(* Logix 5000 project; controller Laser_Cutter vendor 1 type 14 code 149 rev 28.11; software revision 28.00; part 4 of 4 *)
(* tags used below, declared in another part *)
   aAcceptPartSol : BOOL;
   aBlowOffOnSol : BOOL;
   aBoltBowlFeedingOn : BOOL;
   aBoltDriverDownSol : BOOL;
   aBoltDriverForward : BOOL;
   aBoltDriverReverse : BOOL;
   aBoltDriverUpSol : BOOL;
   aBoltFeedingTrackOn : BOOL;
   aCameraTrigger : BOOL;
   acceptPartSol : BOOL;
   aClampingStation2Down : BOOL;
   aClampingStation2Up : BOOL;
   aClampingStation4DownSol : BOOL;
   aClampingStation5DownSol : BOOL;
   aClampingStation5UpSol : BOOL;
   aCollarBowlFeedingOn : BOOL;
   aCollarFeedingTrackOn : BOOL;
   aDoorSafetySwitchUnlockSol : BOOL;
   alarmActive : BOOL;
   aRejectPartSol : BOOL;
   aTapForward : BOOL;
   aTapReverse : BOOL;
   automaticSeqStep : DINT;
   autoMode : BOOL;
   autoModeReady : BOOL;
   aWalkingBeamDownSol : BOOL;
   aWalkingBeamLeftSol : BOOL;
   aWalkingBeamRightSol : BOOL;
   aWalkingBeamUpSol : BOOL;
   boltBowlFeedingOn : BOOL;
   boltDriverDownSol : BOOL;
   boltDriverForward : BOOL;
   boltDriverReverse : BOOL;
   boltDriverUpSol : BOOL;
   cameraTriggerFlag : BOOL;
   cameraTriggerPulse : TIMER;
   clampingStation2Down : BOOL;
   clampingStation2Up : BOOL;
   clampingStation4DownSol : BOOL;
   clampingStation4UpSol : BOOL;
   clampingStation5DownSol : BOOL;
   clampingStation5Sol : BOOL;
   collarBowlFeedingOn : BOOL;
   CYCLE_COMPLETE : BOOL;
   CYCLE_IN_PROG : BOOL;
   cycleTimeBufferMin : DINT;
   cycleTimeBufferSec : DINT;
   cycleTimer : TIMER;
   doorLockAtInitialPosition : BOOL;
   Exec_Tapping_SR : BOOL;
   HMI_AutoMode_Req : BOOL;
   HMI_ManualMode_Req : BOOL;
   idleTime : TIMER;
   idleTimeBufferMin : DINT;
   idleTimeBufferSec : DINT;
   INIT_IN_PROG : BOOL;
   Initialize_Timer : TIMER;
   initSeqStep : DINT;
   lampTestActive : BOOL;
   lampTestPB : BOOL;
   lampTestTimer : TIMER;
   mAcceptPartPB : BOOL;
   mAcceptPartSol : BOOL;
   manualMode : BOOL;
   maTapReversePB : BOOL;
   mBlowOffOn : BOOL;
   mBlowOffOnSol : BOOL;
   mBlowOffSol : BOOL;
   mBoltBowlFeedingOnPB : BOOL;
   mBoltDriverDownPB : BOOL;
   mBoltDriverDownSol : BOOL;
   mBoltDriverForward : BOOL;
   mBoltDriverForwardPB : BOOL;
   mBoltDriverReverse : BOOL;
   mBoltDriverReversePB : BOOL;
   mBoltDriverUpPB : BOOL;
   mBoltDriverUpSol : BOOL;
   mBoltFeedingTrackOnPB : BOOL;
   mcameraTrigger : BOOL;
   mClampingStation2Down : BOOL;
   mClampingStation2DownSol : BOOL;
   mClampingStation2Up : BOOL;
   mClampingStation2UpPB : BOOL;
   mClampingStation2UpSol : BOOL;
   mClampingStation4DownSol : BOOL;
   mClampingStation4UpPB : BOOL;
   mClampingStation4UpSol : BOOL;
   mClampingStation5DownPB : BOOL;
   mClampingStation5DownSol : BOOL;
   mClampingStation5UpPB : BOOL;
   mClampingStation5UpSol : BOOL;
   mClampStation4DownPB : BOOL;
   mCollarBowlFeedingOnPB : BOOL;
   mCollarFeedingTrackOnPB : BOOL;
   mDoorSafetySwitchUnlockSol : BOOL;
   mRejectPartPB : BOOL;
   mRejectPartSol : BOOL;
   mTapForward : BOOL;
   mTapForwardPB : BOOL;
   mTapReverse : BOOL;
   mWalkingBeamDownPB : BOOL;
   mWalkingBeamDownSol : BOOL;
   mWalkingBeamLeftPB : BOOL;
   mWalkingBeamLeftSol : BOOL;
   mWalkingBeamRightPB : BOOL;
   mWalkingBeamRightSol : BOOL;
   mWalkingBeamUpPB : BOOL;
   mWalkingBeamUpSol : BOOL;
   p2pCycleTimeBuffer : DINT;
   p2pCycleTimeBufferSec : DINT;
   rejectPartSol : BOOL;
   resetPartCountingValuesHMIPB : BOOL;
   resetPartCountingValuesTimer : TIMER;
   runTime : TIMER;
   runTimeBufferMin : DINT;
   runTimeBufferSec : DINT;
   tapDownDB : TIMER;
   tapUpDB : TIMER;
   TMR_PULSE_OFF : TIMER;
   TMR_PULSE_ON : TIMER;
   walkingBeamDownSol : BOOL;
   walkingBeamLeftSol : BOOL;
   walkingBeamRightSol : BOOL;
   walkingBeamUpSol : BOOL;
   blowOffOn : ALIAS FOR Local:1:O.Data.9;
   boltFeedingTrackOn : ALIAS FOR Local:1:O.Data.8;
   cameraTrigger : ALIAS FOR Local:1:O.Data.11;
   collarFeedingTrackOn : ALIAS FOR Local:1:O.Data.6;
   currentUser : DINT;   // Access Level of current user
   doorSafetySwitchUnlockSol : ALIAS FOR Local:1:O.Data.10;
   greenStatusLight : ALIAS FOR Local:1:O.Data.2;
   redStatusLight : ALIAS FOR Local:1:O.Data.0;
   tapForward : ALIAS FOR MURR_IMPACT_IO_2:O.Data[0].0;
   tapReverse : ALIAS FOR MURR_IMPACT_IO_2:O.Data[0].1;
   yellowStatusLight : ALIAS FOR Local:1:O.Data.1;
(* MainProgram, continued *)

ROUTINE MainRoutine   (* ladder *)
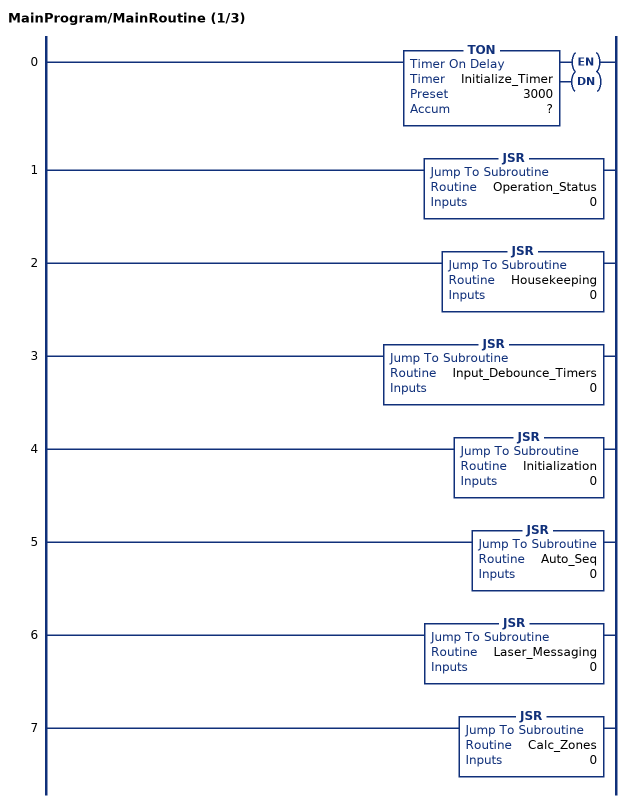
   0: TON(Initialize_Timer,?,?);
   1: JSR(Operation_Status,0);
   2: JSR(Housekeeping,0);
   3: JSR(Input_Debounce_Timers,0);
   4: JSR(Initialization,0);
   5: JSR(Auto_Seq,0);
   6: JSR(Laser_Messaging,0);
   7: JSR(Calc_Zones,0);
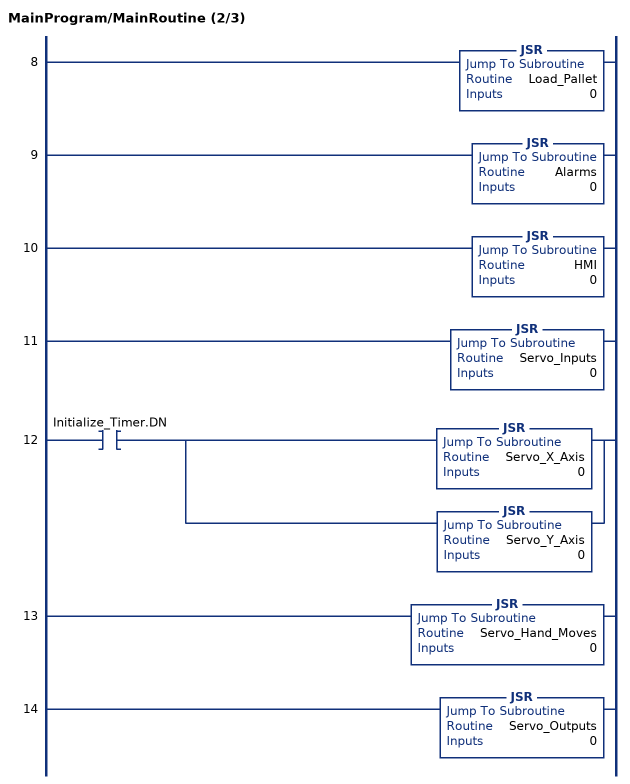
   8: JSR(Load_Pallet,0);
   9: JSR(Alarms,0);
   10: JSR(HMI,0);
   11: JSR(Servo_Inputs,0);
   12: XIC(Initialize_Timer.DN)[JSR(Servo_X_Axis,0) ,JSR(Servo_Y_Axis,0) ];
   13: JSR(Servo_Hand_Moves,0);
   14: JSR(Servo_Outputs,0);
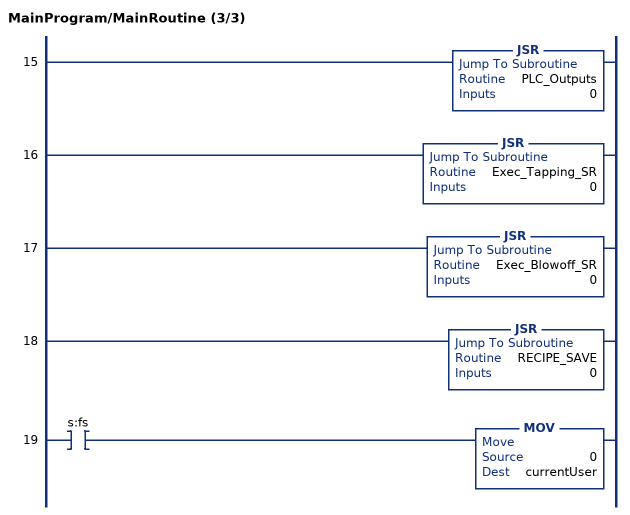
   15: JSR(PLC_Outputs,0);
   16: JSR(Exec_Tapping_SR,0);
   17: JSR(Exec_Blowoff_SR,0);
   18: JSR(RECIPE_SAVE,0);
   19: XIC(s:fs)MOV(0,currentUser);
END_ROUTINE

ROUTINE Operation_Status   (* ladder *)
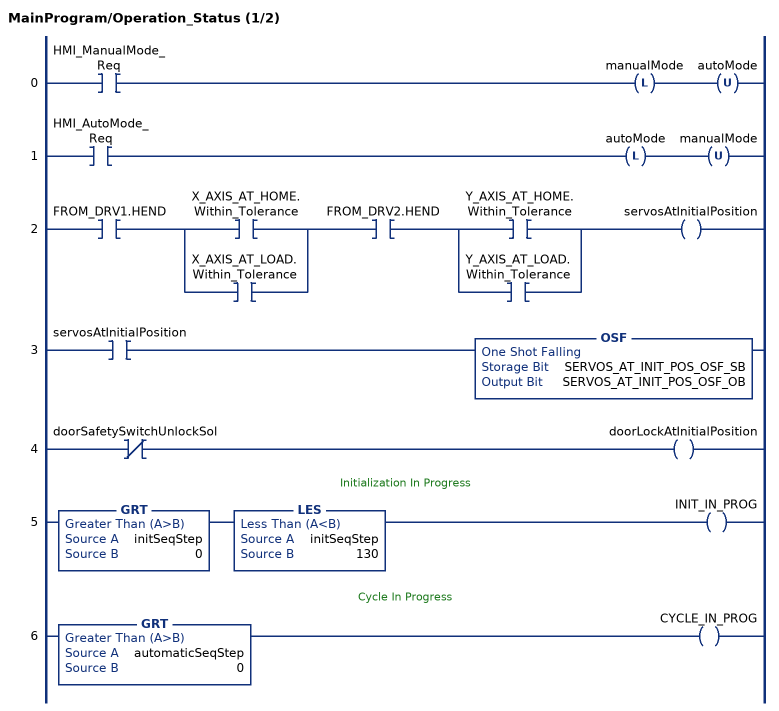
   0: XIC(HMI_ManualMode_Req)OTL(manualMode)OTU(autoMode);
   1: XIC(HMI_AutoMode_Req)OTL(autoMode)OTU(manualMode);
   2: XIC(FROM_DRV1.HEND)[XIC(X_AXIS_AT_HOME.Within_Tolerance) ,XIC(X_AXIS_AT_LOAD.Within_Tolerance) ]XIC(FROM_DRV2.HEND)[XIC(Y_AXIS_AT_HOME.Within_Tolerance) ,XIC(Y_AXIS_AT_LOAD.Within_Tolerance) ]OTE(servosAtInitialPosition);
   3: XIC(servosAtInitialPosition)OSF(SERVOS_AT_INIT_POS_OSF_SB,SERVOS_AT_INIT_POS_OSF_OB);
   4: XIO(doorSafetySwitchUnlockSol)OTE(doorLockAtInitialPosition);
   // Initialization In Progress
   5: GRT(initSeqStep,0)LES(initSeqStep,130)OTE(INIT_IN_PROG);
   // Cycle In Progress
   6: GRT(automaticSeqStep,0)OTE(CYCLE_IN_PROG);
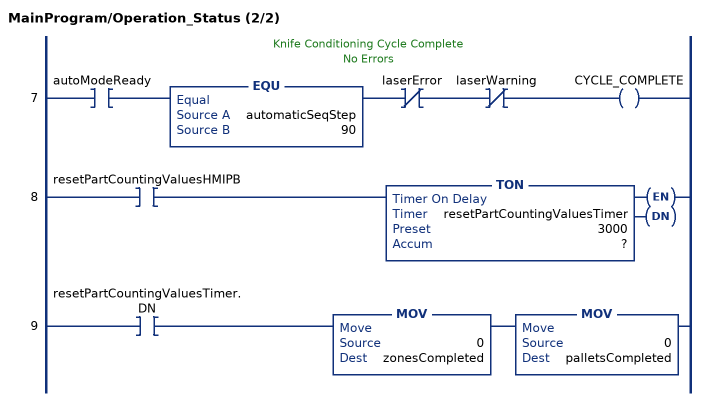
   // Knife Conditioning Cycle Complete
   // No Errors
   7: XIC(autoModeReady)EQU(automaticSeqStep,90)XIO(laserError)XIO(laserWarning)OTE(CYCLE_COMPLETE);
   8: XIC(resetPartCountingValuesHMIPB)TON(resetPartCountingValuesTimer,?,?);
   9: XIC(resetPartCountingValuesTimer.DN)MOV(0,zonesCompleted)MOV(0,palletsCompleted);
END_ROUTINE

ROUTINE PLC_Outputs   (* ladder *)
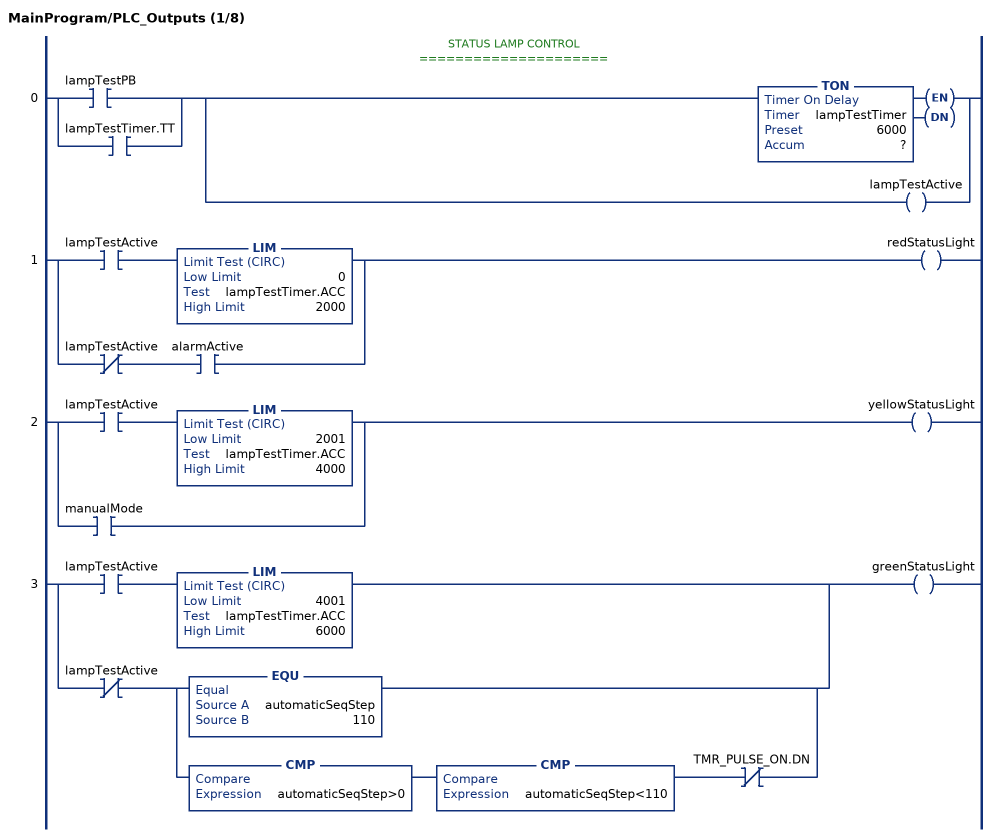
   // STATUS LAMP CONTROL
   // =====================
   0: [XIC(lampTestPB) ,XIC(lampTestTimer.TT) ][TON(lampTestTimer,?,?) ,OTE(lampTestActive) ];
   1: [XIC(lampTestActive) LIM(0,lampTestTimer.ACC,2000) ,XIO(lampTestActive) XIC(alarmActive) ]OTE(redStatusLight);
   2: [XIC(lampTestActive) LIM(2001,lampTestTimer.ACC,4000) ,XIC(manualMode) ]OTE(yellowStatusLight);
   3: [XIC(lampTestActive) LIM(4001,lampTestTimer.ACC,6000) ,XIO(lampTestActive) [EQU(automaticSeqStep,110) ,CMP(automaticSeqStep>0) CMP(automaticSeqStep<110) XIO(TMR_PULSE_ON.DN) ] ]OTE(greenStatusLight);
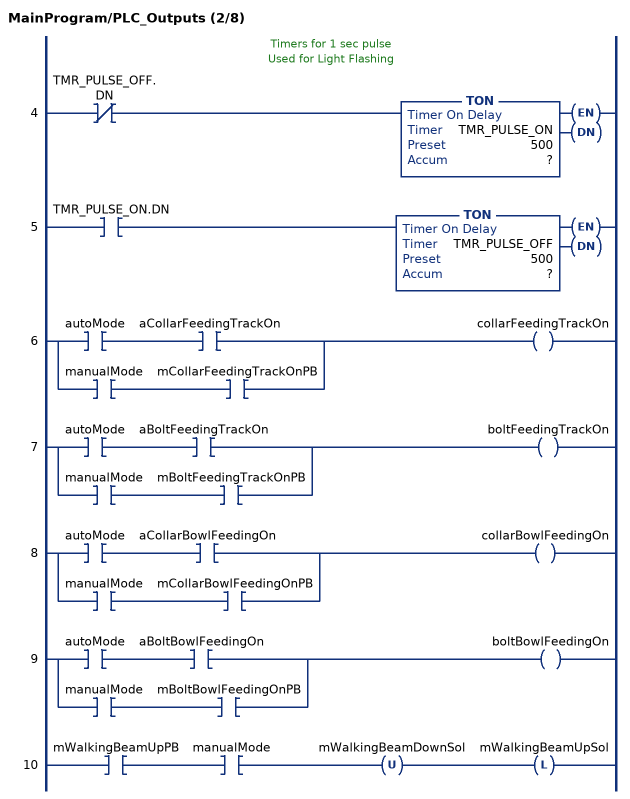
   // Timers for 1 sec pulse
   // Used for Light Flashing
   4: XIO(TMR_PULSE_OFF.DN)TON(TMR_PULSE_ON,?,?);
   5: XIC(TMR_PULSE_ON.DN)TON(TMR_PULSE_OFF,?,?);
   6: [XIC(autoMode) XIC(aCollarFeedingTrackOn) ,XIC(manualMode) XIC(mCollarFeedingTrackOnPB) ]OTE(collarFeedingTrackOn);
   7: [XIC(autoMode) XIC(aBoltFeedingTrackOn) ,XIC(manualMode) XIC(mBoltFeedingTrackOnPB) ]OTE(boltFeedingTrackOn);
   8: [XIC(autoMode) XIC(aCollarBowlFeedingOn) ,XIC(manualMode) XIC(mCollarBowlFeedingOnPB) ]OTE(collarBowlFeedingOn);
   9: [XIC(autoMode) XIC(aBoltBowlFeedingOn) ,XIC(manualMode) XIC(mBoltBowlFeedingOnPB) ]OTE(boltBowlFeedingOn);
   10: XIC(mWalkingBeamUpPB)XIC(manualMode)OTU(mWalkingBeamDownSol)OTL(mWalkingBeamUpSol);
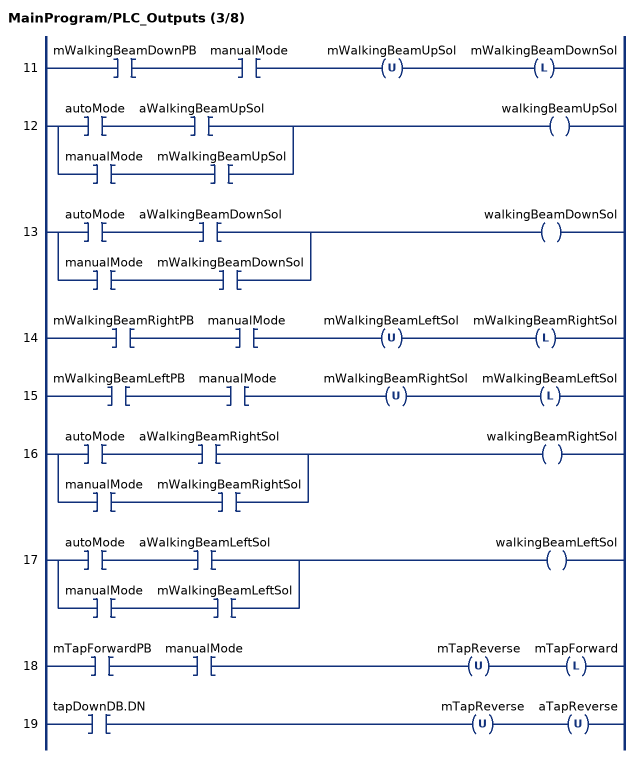
   11: XIC(mWalkingBeamDownPB)XIC(manualMode)OTU(mWalkingBeamUpSol)OTL(mWalkingBeamDownSol);
   12: [XIC(autoMode) XIC(aWalkingBeamUpSol) ,XIC(manualMode) XIC(mWalkingBeamUpSol) ]OTE(walkingBeamUpSol);
   13: [XIC(autoMode) XIC(aWalkingBeamDownSol) ,XIC(manualMode) XIC(mWalkingBeamDownSol) ]OTE(walkingBeamDownSol);
   14: XIC(mWalkingBeamRightPB)XIC(manualMode)OTU(mWalkingBeamLeftSol)OTL(mWalkingBeamRightSol);
   15: XIC(mWalkingBeamLeftPB)XIC(manualMode)OTU(mWalkingBeamRightSol)OTL(mWalkingBeamLeftSol);
   16: [XIC(autoMode) XIC(aWalkingBeamRightSol) ,XIC(manualMode) XIC(mWalkingBeamRightSol) ]OTE(walkingBeamRightSol);
   17: [XIC(autoMode) XIC(aWalkingBeamLeftSol) ,XIC(manualMode) XIC(mWalkingBeamLeftSol) ]OTE(walkingBeamLeftSol);
   18: XIC(mTapForwardPB)XIC(manualMode)OTU(mTapReverse)OTL(mTapForward);
   19: XIC(tapDownDB.DN)OTU(mTapReverse)OTU(aTapReverse);
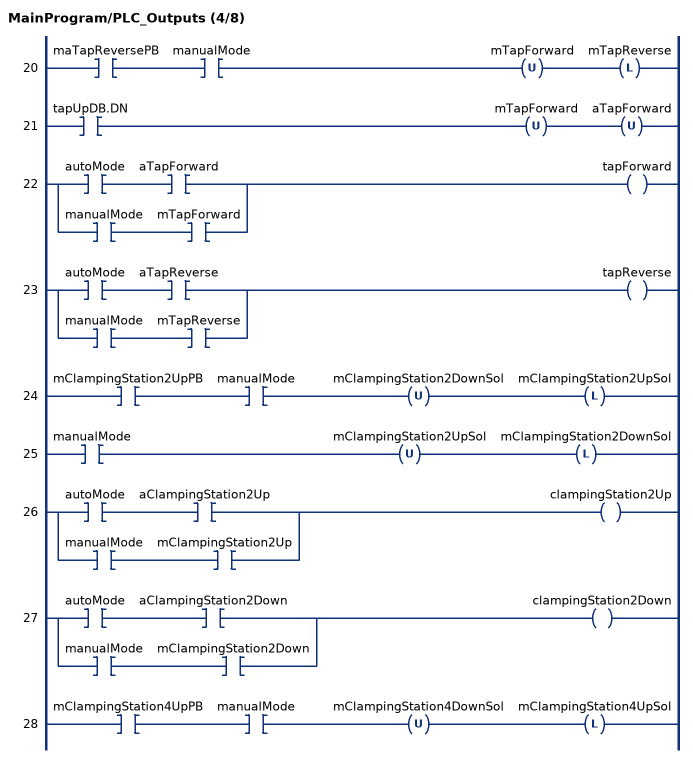
   20: XIC(maTapReversePB)XIC(manualMode)OTU(mTapForward)OTL(mTapReverse);
   21: XIC(tapUpDB.DN)OTU(mTapForward)OTU(aTapForward);
   22: [XIC(autoMode) XIC(aTapForward) ,XIC(manualMode) XIC(mTapForward) ]OTE(tapForward);
   23: [XIC(autoMode) XIC(aTapReverse) ,XIC(manualMode) XIC(mTapReverse) ]OTE(tapReverse);
   24: XIC(mClampingStation2UpPB)XIC(manualMode)OTU(mClampingStation2DownSol)OTL(mClampingStation2UpSol);
   25: XIC(manualMode)OTU(mClampingStation2UpSol)OTL(mClampingStation2DownSol);
   26: [XIC(autoMode) XIC(aClampingStation2Up) ,XIC(manualMode) XIC(mClampingStation2Up) ]OTE(clampingStation2Up);
   27: [XIC(autoMode) XIC(aClampingStation2Down) ,XIC(manualMode) XIC(mClampingStation2Down) ]OTE(clampingStation2Down);
   28: XIC(mClampingStation4UpPB)XIC(manualMode)OTU(mClampingStation4DownSol)OTL(mClampingStation4UpSol);
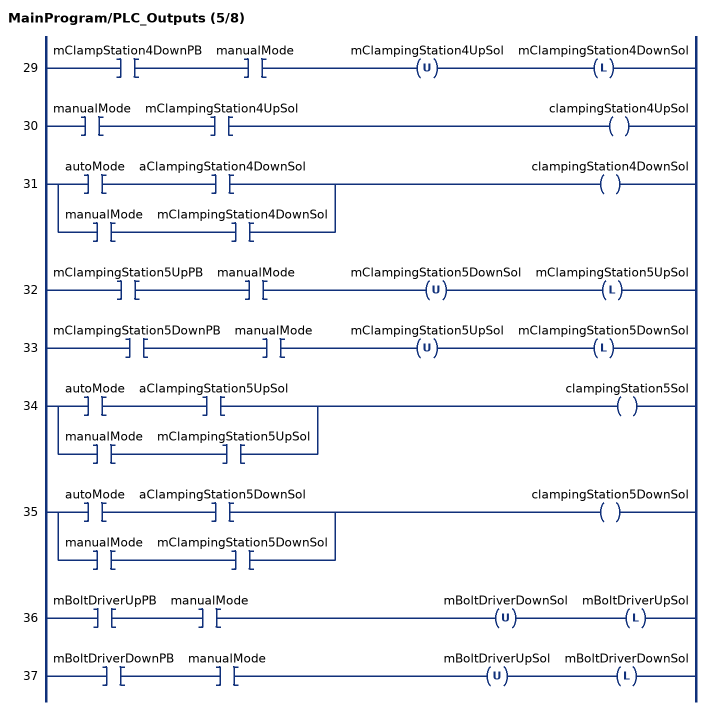
   29: XIC(mClampStation4DownPB)XIC(manualMode)OTU(mClampingStation4UpSol)OTL(mClampingStation4DownSol);
   30: XIC(manualMode)XIC(mClampingStation4UpSol)OTE(clampingStation4UpSol);
   31: [XIC(autoMode) XIC(aClampingStation4DownSol) ,XIC(manualMode) XIC(mClampingStation4DownSol) ]OTE(clampingStation4DownSol);
   32: XIC(mClampingStation5UpPB)XIC(manualMode)OTU(mClampingStation5DownSol)OTL(mClampingStation5UpSol);
   33: XIC(mClampingStation5DownPB)XIC(manualMode)OTU(mClampingStation5UpSol)OTL(mClampingStation5DownSol);
   34: [XIC(autoMode) XIC(aClampingStation5UpSol) ,XIC(manualMode) XIC(mClampingStation5UpSol) ]OTE(clampingStation5Sol);
   35: [XIC(autoMode) XIC(aClampingStation5DownSol) ,XIC(manualMode) XIC(mClampingStation5DownSol) ]OTE(clampingStation5DownSol);
   36: XIC(mBoltDriverUpPB)XIC(manualMode)OTU(mBoltDriverDownSol)OTL(mBoltDriverUpSol);
   37: XIC(mBoltDriverDownPB)XIC(manualMode)OTU(mBoltDriverUpSol)OTL(mBoltDriverDownSol);
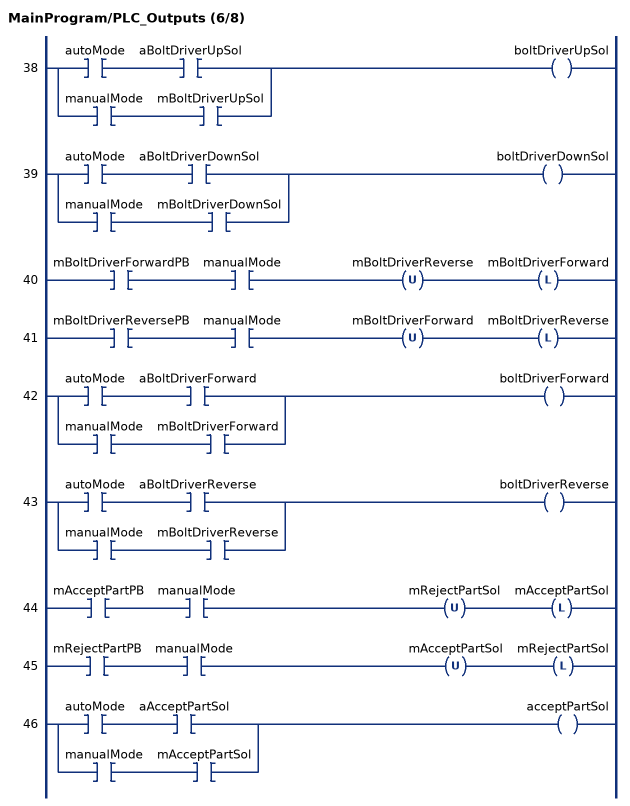
   38: [XIC(autoMode) XIC(aBoltDriverUpSol) ,XIC(manualMode) XIC(mBoltDriverUpSol) ]OTE(boltDriverUpSol);
   39: [XIC(autoMode) XIC(aBoltDriverDownSol) ,XIC(manualMode) XIC(mBoltDriverDownSol) ]OTE(boltDriverDownSol);
   40: XIC(mBoltDriverForwardPB)XIC(manualMode)OTU(mBoltDriverReverse)OTL(mBoltDriverForward);
   41: XIC(mBoltDriverReversePB)XIC(manualMode)OTU(mBoltDriverForward)OTL(mBoltDriverReverse);
   42: [XIC(autoMode) XIC(aBoltDriverForward) ,XIC(manualMode) XIC(mBoltDriverForward) ]OTE(boltDriverForward);
   43: [XIC(autoMode) XIC(aBoltDriverReverse) ,XIC(manualMode) XIC(mBoltDriverReverse) ]OTE(boltDriverReverse);
   44: XIC(mAcceptPartPB)XIC(manualMode)OTU(mRejectPartSol)OTL(mAcceptPartSol);
   45: XIC(mRejectPartPB)XIC(manualMode)OTU(mAcceptPartSol)OTL(mRejectPartSol);
   46: [XIC(autoMode) XIC(aAcceptPartSol) ,XIC(manualMode) XIC(mAcceptPartSol) ]OTE(acceptPartSol);
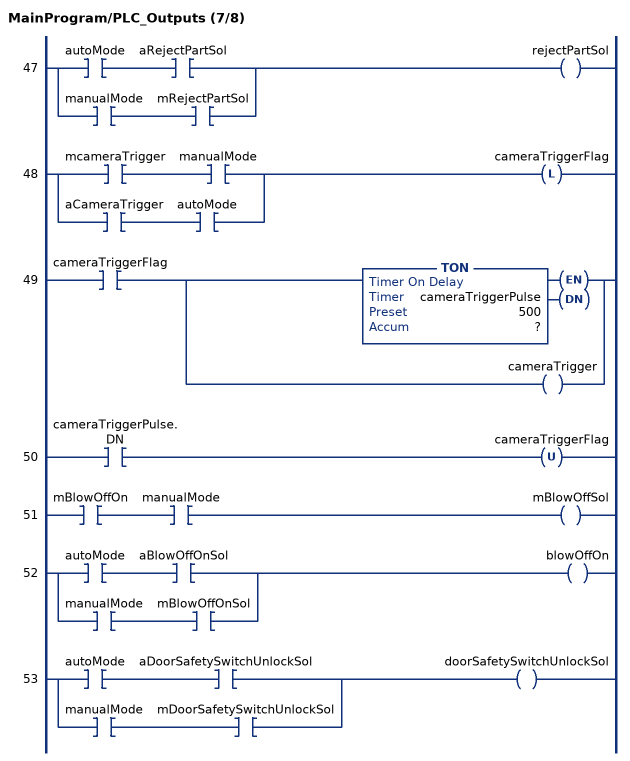
   47: [XIC(autoMode) XIC(aRejectPartSol) ,XIC(manualMode) XIC(mRejectPartSol) ]OTE(rejectPartSol);
   48: [XIC(mcameraTrigger) XIC(manualMode) ,XIC(aCameraTrigger) XIC(autoMode) ]OTL(cameraTriggerFlag);
   49: XIC(cameraTriggerFlag)[TON(cameraTriggerPulse,?,?) ,OTE(cameraTrigger) ];
   50: XIC(cameraTriggerPulse.DN)OTU(cameraTriggerFlag);
   51: XIC(mBlowOffOn)XIC(manualMode)OTE(mBlowOffSol);
   52: [XIC(autoMode) XIC(aBlowOffOnSol) ,XIC(manualMode) XIC(mBlowOffOnSol) ]OTE(blowOffOn);
   53: [XIC(autoMode) XIC(aDoorSafetySwitchUnlockSol) ,XIC(manualMode) XIC(mDoorSafetySwitchUnlockSol) ]OTE(doorSafetySwitchUnlockSol);
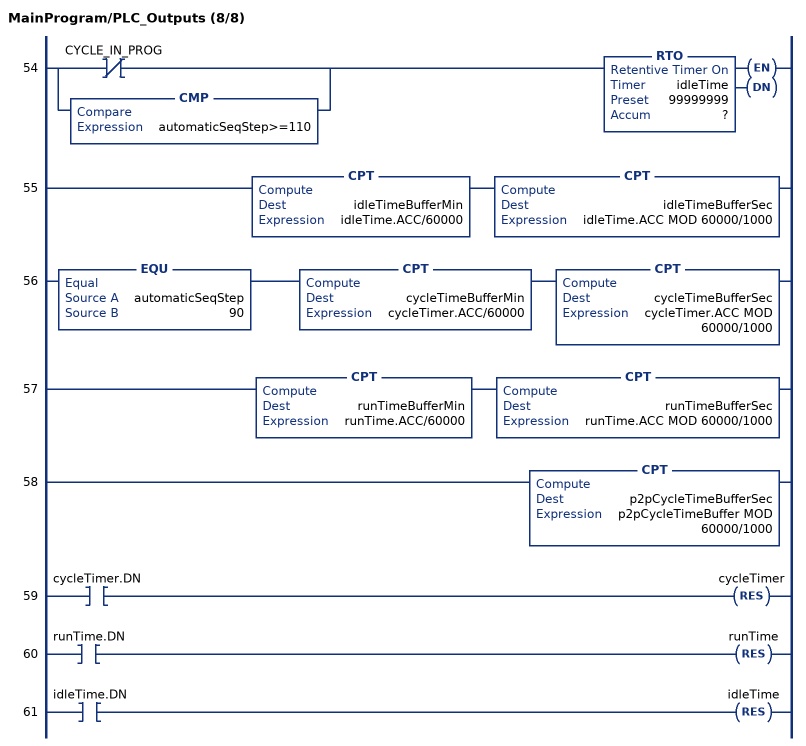
   54: [XIO(CYCLE_IN_PROG) ,CMP(automaticSeqStep>=110) ]RTO(idleTime,?,?);
   55: CPT(idleTimeBufferMin,idleTime.ACC/60000)CPT(idleTimeBufferSec,idleTime.ACC MOD 60000/1000);
   56: EQU(automaticSeqStep,90)CPT(cycleTimeBufferMin,cycleTimer.ACC/60000)CPT(cycleTimeBufferSec,cycleTimer.ACC MOD 60000/1000);
   57: CPT(runTimeBufferMin,runTime.ACC/60000)CPT(runTimeBufferSec,runTime.ACC MOD 60000/1000);
   58: CPT(p2pCycleTimeBufferSec,p2pCycleTimeBuffer MOD 60000/1000);
   59: XIC(cycleTimer.DN)RES(cycleTimer);
   60: XIC(runTime.DN)RES(runTime);
   61: XIC(idleTime.DN)RES(idleTime);
END_ROUTINE
END_PROGRAM
